(*

## Short summary

This class provides assert statements for strings
For UTF-16 strings up to 255 ``WORD`` (``WSTRING(Tc2_System.MAX_STRING_LENGTH)``) use the property `IStringAssertions.utf16`.
For windows-1252 strings up to 255 ``BYTE`` (``Tc2_System.T_MaxString``) use the property `IStringAssertions.windows1252`.
For windows-1252 or UTF-16 strings that are longer, use the property `IStringAssertions.anyString`  

.. <legal notes>

legal notes
=================
| SPDX-FileCopyrightText: © 2022 ekvip automation GmbH <info@ekvip.de>
| SPDX-License-Identifier: Apache-2.0
| For details check: Apache-2.0_

.. _Apache-2.0: https://www.apache.org/licenses/LICENSE-2.0

.. </legal notes>



*)

{attribute 'reflection'}
FUNCTION_BLOCK INTERNAL StringAssertions EXTENDS CNM_AbstractObject.Object IMPLEMENTS IStringAssertions, IAssertCallBackSetter
VAR
	(* class to handle windows-1252 and windows-1251 assertions *)
	win125xStringAssertions	:Windows125xStringAssertions();
	(* class to handle UTF-16 assertions *)
	utf16StringAssertions	:Utf16StringAssertions();
	(* class to handle UTF-8 assertions *)
	utf8StringAssertions	:Utf8StringAssertions();
	(* class to handle Unicode assertions with anys string*)
	UnicodeAssertions :UnicodeAssertions();
END_VAR

(*

## Short summary
This abstract property returns the class name of the concrete object, 
It's for debugging purpose

.. <legal notes>

legal notes
=================
| SPDX-FileCopyrightText: © 2022 ekvip automation GmbH <info@ekvip.de>
| SPDX-License-Identifier: Apache-2.0
| For details check: Apache-2.0_

.. _Apache-2.0: https://www.apache.org/licenses/LICENSE-2.0

.. </legal notes>

*)

PROPERTY className :CNM_AbstractObject.ClassName
GET
className := 'CNM_Assertor.StringAssertions';
END_GET
END_PROPERTY

(*

## Short summary
This methods is the setter for the callback class if an assertion was false

.. <legal notes>

legal notes
=================
| SPDX-FileCopyrightText: © 2022 ekvip automation GmbH <info@ekvip.de>
| SPDX-License-Identifier: Apache-2.0
| For details check: Apache-2.0_

.. _Apache-2.0: https://www.apache.org/licenses/LICENSE-2.0

.. </legal notes>



*)

METHOD setCallBack
VAR_INPUT
	(* the class that must be informed if an assertion is false *)
	callBack	: IAssertCallBack;
END_VAR
THIS^.utf16StringAssertions.setCallBack(callBack);
THIS^.win125xStringAssertions.setCallBack(callBack);
THIS^.utf8StringAssertions.setCallBack(callBack);
THIS^.UnicodeAssertions.setCallBack(callBack);
END_METHOD

(*

## Short summary
Returns an interface `IUnicodeStringAssertions` with assert statements,
for UTF-8 and UTF-16 strings with an undefined length.

**Attention:** 
	All strings are handled as null terminated byte/word streams.
	For UTF-8 is end of the string 16#00
	For UTF-16 is end of the string 16#00_00

**Attention:** 
	The interface `IUnicodeAssertions` uses ``ANY_STRING``, 
	for this it's not possible to use literals/constants,
	because for ``ANY`` types generates the compiler ``__SYSTEM.AnyType``
	and ``__SYSTEM.AnyType`` contains a pointer  

.. <legal notes>

legal notes
=================
| SPDX-FileCopyrightText: © 2022 ekvip automation GmbH <info@ekvip.de>
| SPDX-License-Identifier: Apache-2.0
| For details check: Apache-2.0_

.. _Apache-2.0: https://www.apache.org/licenses/LICENSE-2.0

.. </legal notes>

*)
PROPERTY unicode :IUnicodeStringAssertions
GET
unicode := THIS^.UnicodeAssertions;
END_GET
END_PROPERTY

(*

## Short summary
Returns an interface `IUtf16StringAssertions` with assert statements
for UTF-16 strings until 255 ``WORD`` length (``WSTRING(Tc2_System.MAX_STRING_LENGTH)``)

.. <legal notes>

legal notes
=================
| SPDX-FileCopyrightText: © 2022 ekvip automation GmbH <info@ekvip.de>
| SPDX-License-Identifier: Apache-2.0
| For details check: Apache-2.0_

.. _Apache-2.0: https://www.apache.org/licenses/LICENSE-2.0

.. </legal notes>

*)

PROPERTY utf16 :IUtf16StringAssertions
GET
utf16 := THIS^.utf16StringAssertions;
END_GET
END_PROPERTY

(*

## Short summary
Returns an interface `IUtf8StringAssertions` with assert statements
for UTF-8 strings up to 255 bytes length (``STRING(Tc2_System.MAX_STRING_LENGTH)``)

.. <legal notes>

legal notes
=================
| SPDX-FileCopyrightText: © 2022 ekvip automation GmbH <info@ekvip.de>
| SPDX-License-Identifier: Apache-2.0
| For details check: Apache-2.0_

.. _Apache-2.0: https://www.apache.org/licenses/LICENSE-2.0

.. </legal notes>

*)

PROPERTY utf8 :IUtf8StringAssertions
GET
utf8 := THIS^.utf8StringAssertions;
END_GET
END_PROPERTY

(*

## Short summary
Returns an interface `IWindows125xStringAssertions` with assert statements for 8-bit 
windows-1252 and windows-1251 strings up to 255 characters length (``Tc2_System.T_MaxString``).
Use Tc2_Utilities.GLOBAL_SBCS_TABLE variable to select required encoding

.. <legal notes>

legal notes
=================
| SPDX-FileCopyrightText: © 2022 ekvip automation GmbH <info@ekvip.de>
| SPDX-License-Identifier: Apache-2.0
| For details check: Apache-2.0_

.. _Apache-2.0: https://www.apache.org/licenses/LICENSE-2.0

.. </legal notes>

*)

PROPERTY windows125x :IWindows125xStringAssertions
GET
windows125x := THIS^.win125xStringAssertions;
END_GET
END_PROPERTY

END_FUNCTION_BLOCK

(* stored: Version 1.1.0.1, ProductVersion 3.1.4026.12
   POU StringAssertions: Id {021e2eff-f314-4410-aa94-a992b4891e84}, SpecialFunc None
   Property className: Id {555ec8d0-998c-4d51-947b-a00038fc251b}
   Get Get: Id {e2549954-2db4-4937-90fc-d9afd1f6530d}
   Method setCallBack: Id {98d51a66-31a8-4e14-8d43-1c3d68f8920a}
   Property unicode: Id {9c482a1e-ec38-4ab4-a917-d8c37a173922}
   Get Get: Id {20d81158-4ead-47e2-b859-1b8aa91f45c9}
   Property utf16: Id {8c35efe3-da80-4ce5-b25e-cf1d715e4a32}
   Get Get: Id {b900738d-a5d9-4419-bc9c-6054032e3597}
   Property utf8: Id {68e05729-c5c3-436c-9817-db5dd5fb6dd9}
   Get Get: Id {14904fa8-0041-490e-8625-75b8c18023a2}
   Property windows125x: Id {4708f9dd-1d22-44f6-bc75-c94afb229506}
   Get Get: Id {079a5602-99f9-4f76-b15a-05247b62e830} *)
